% RSLogix 500 project I2P JOB 15_RUSSELL_BAK014.RSS, saved by version 10.00.00.00 %
PROJECT "ML02A"    % processor: Bul.1763 MicroLogix 1100 Series B %

PROGRAM FILES
  LAD 2   13 rungs

DATA FILES
  O0 OUTPUT  4 elements
  I1 INPUT  6 elements
  S2 STATUS  66 elements
  B3 BINARY  1 elements
  T4 TIMER  2 elements
  C5 COUNTER  1 elements
  R6 CONTROL  1 elements
  N7 INTEGER  1 elements
  F8 FLOAT  1 elements

LADDER 2
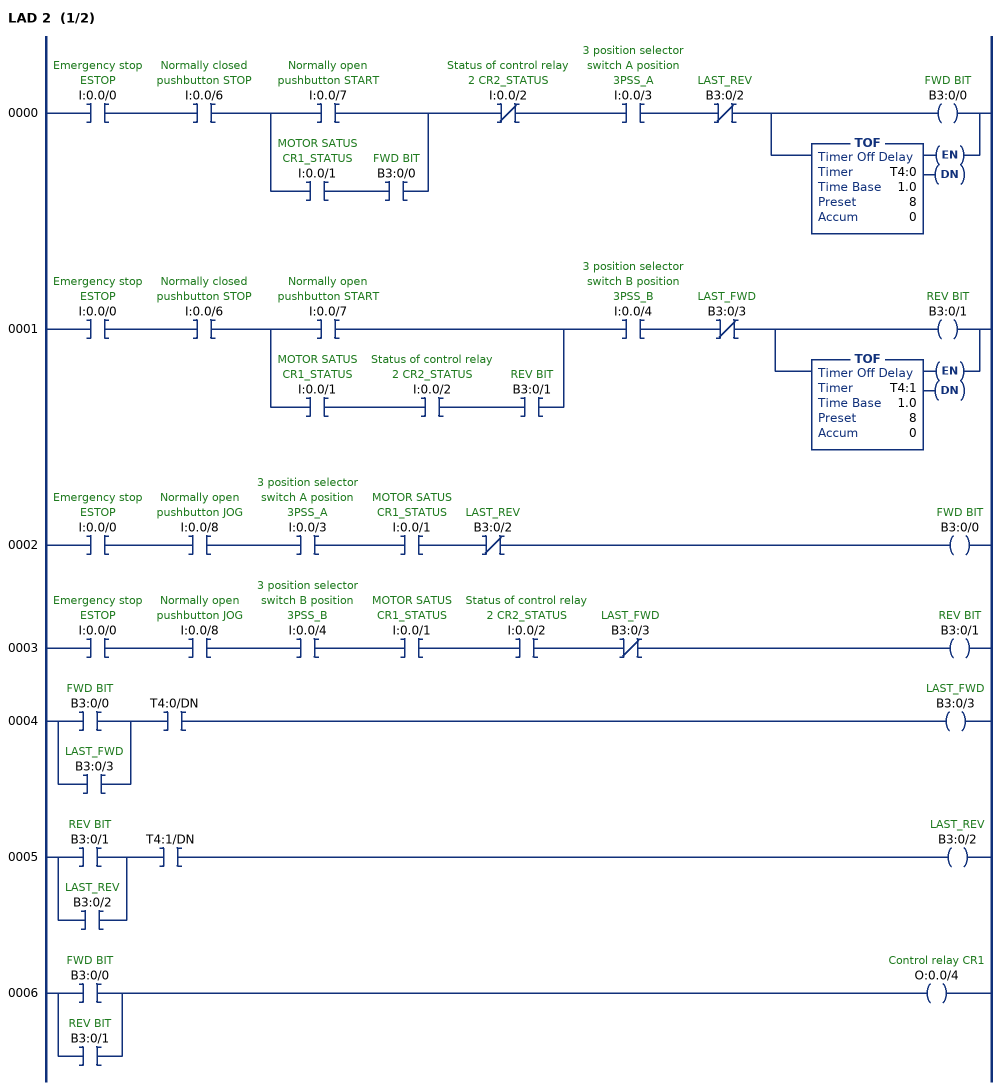
% Rung: 0 %
SOR XIC I:0.0/0 XIC I:0.0/6 BST XIC I:0.0/7 NXB XIC I:0.0/1 XIC B3:0/0 BND XIO I:0.0/2 XIC I:0.0/3 XIO B3:0/2 BST OTE B3:0/0 NXB TOF T4:0 1.0 8 0 BND EOR
%   I:0.0/0  ESTOP  "Emergency stop" %
%   I:0.0/6  STOP  "Normally closed pushbutton" %
%   I:0.0/7  START  "Normally open pushbutton" %
%   I:0.0/1  CR1_STATUS  "MOTOR SATUS" %
%   B3:0/0  "FWD BIT" %
%   I:0.0/2  CR2_STATUS  "Status of control relay 2" %
%   I:0.0/3  3PSS_A  "3 position selector switch A position" %
%   B3:0/2  LAST_REV %
% Rung: 1 %
SOR XIC I:0.0/0 XIC I:0.0/6 BST XIC I:0.0/7 NXB XIC I:0.0/1 XIC I:0.0/2 XIC B3:0/1 BND XIC I:0.0/4 XIO B3:0/3 BST OTE B3:0/1 NXB TOF T4:1 1.0 8 0 BND EOR
%   I:0.0/0  ESTOP  "Emergency stop" %
%   I:0.0/6  STOP  "Normally closed pushbutton" %
%   I:0.0/7  START  "Normally open pushbutton" %
%   I:0.0/1  CR1_STATUS  "MOTOR SATUS" %
%   I:0.0/2  CR2_STATUS  "Status of control relay 2" %
%   B3:0/1  "REV BIT" %
%   I:0.0/4  3PSS_B  "3 position selector switch B position" %
%   B3:0/3  LAST_FWD %
% Rung: 2 %
SOR XIC I:0.0/0 XIC I:0.0/8 XIC I:0.0/3 XIC I:0.0/1 XIO B3:0/2 OTE B3:0/0 EOR
%   I:0.0/0  ESTOP  "Emergency stop" %
%   I:0.0/8  JOG  "Normally open pushbutton" %
%   I:0.0/3  3PSS_A  "3 position selector switch A position" %
%   I:0.0/1  CR1_STATUS  "MOTOR SATUS" %
%   B3:0/2  LAST_REV %
%   B3:0/0  "FWD BIT" %
% Rung: 3 %
SOR XIC I:0.0/0 XIC I:0.0/8 XIC I:0.0/4 XIC I:0.0/1 XIC I:0.0/2 XIO B3:0/3 OTE B3:0/1 EOR
%   I:0.0/0  ESTOP  "Emergency stop" %
%   I:0.0/8  JOG  "Normally open pushbutton" %
%   I:0.0/4  3PSS_B  "3 position selector switch B position" %
%   I:0.0/1  CR1_STATUS  "MOTOR SATUS" %
%   I:0.0/2  CR2_STATUS  "Status of control relay 2" %
%   B3:0/3  LAST_FWD %
%   B3:0/1  "REV BIT" %
% Rung: 4 %
SOR BST XIC B3:0/0 NXB XIC B3:0/3 BND XIC T4:0/DN OTE B3:0/3 EOR
%   B3:0/0  "FWD BIT" %
%   B3:0/3  LAST_FWD %
% Rung: 5 %
SOR BST XIC B3:0/1 NXB XIC B3:0/2 BND XIC T4:1/DN OTE B3:0/2 EOR
%   B3:0/1  "REV BIT" %
%   B3:0/2  LAST_REV %
% Rung: 6 %
SOR BST XIC B3:0/0 NXB XIC B3:0/1 BND OTE O:0.0/4 EOR
%   B3:0/0  "FWD BIT" %
%   B3:0/1  "REV BIT" %
%   O:0.0/4  CR1  "Control relay" %

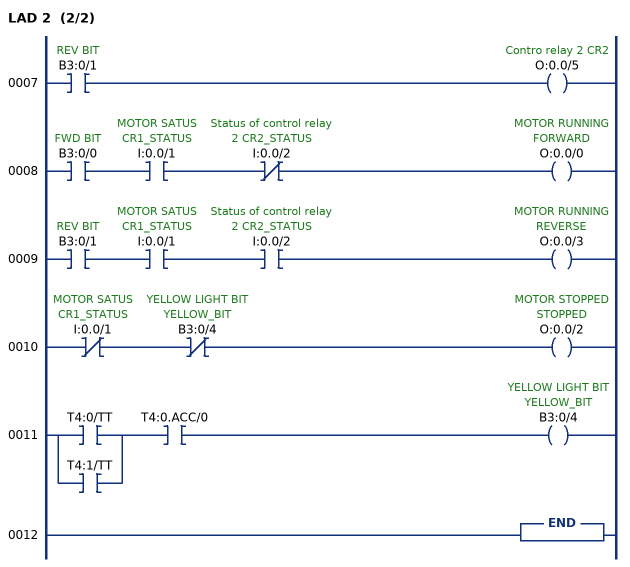
% Rung: 7 %
SOR XIC B3:0/1 OTE O:0.0/5 EOR
%   B3:0/1  "REV BIT" %
%   O:0.0/5  CR2  "Contro relay 2" %
% Rung: 8 %
SOR XIC B3:0/0 XIC I:0.0/1 XIO I:0.0/2 OTE O:0.0/0 EOR
%   B3:0/0  "FWD BIT" %
%   I:0.0/1  CR1_STATUS  "MOTOR SATUS" %
%   I:0.0/2  CR2_STATUS  "Status of control relay 2" %
%   O:0.0/0  FORWARD  "MOTOR RUNNING" %
% Rung: 9 %
SOR XIC B3:0/1 XIC I:0.0/1 XIC I:0.0/2 OTE O:0.0/3 EOR
%   B3:0/1  "REV BIT" %
%   I:0.0/1  CR1_STATUS  "MOTOR SATUS" %
%   I:0.0/2  CR2_STATUS  "Status of control relay 2" %
%   O:0.0/3  REVERSE  "MOTOR RUNNING" %
% Rung: 10 %
SOR XIO I:0.0/1 XIO B3:0/4 OTE O:0.0/2 EOR
%   I:0.0/1  CR1_STATUS  "MOTOR SATUS" %
%   B3:0/4  YELLOW_BIT  "YELLOW LIGHT BIT" %
%   O:0.0/2  STOPPED  "MOTOR STOPPED" %
% Rung: 11 %
SOR BST XIC T4:0/TT NXB XIC T4:1/TT BND XIC T4:0.ACC/0 OTE B3:0/4 EOR
%   B3:0/4  YELLOW_BIT  "YELLOW LIGHT BIT" %
% Rung: 12 %
SOR END EOR

OTHER DOCUMENTED ADDRESSES
  I:0.0/5  RUN_JOG  "Run/Jog Mode (A = Run, B - Jog)"
  O:0.0/1  YELLOW_LIGHT  "Yellow light"

DATA TABLE (non-zero values as saved)
DATA T4
% .PRE .ACC %
% T4:0 % 8 0
% T4:1 % 8 0
DATA C5
% .PRE .ACC %
% C5:0 % 16 8
